Staubli VAL3: recvHeartbeat.pgx

public program recvHeartbeat()
  local num l_nByte
  local num l_nBytesRecv
  local num l_nHtbt
  local num l_nHtbtB[4]
  local num l_nIndex
begin
  while (true)
    l_nBytesRecv=0
    l_nIndex=0
    // if heartbeat is expected (used with mock client)
    if (bCheckHeartbeat)
      // attempt to receive heartbeat
      while (l_nBytesRecv<4)
        l_nIndex=sioGet(siTcpIpFbk,l_nByte)
        if (l_nIndex==1)
          l_nHtbtB[l_nBytesRecv]=l_nByte
          l_nBytesRecv=l_nBytesRecv+l_nIndex
        elseIf (l_nIndex==-1)
          // error or timeout, indicate only if connection previously established
          if (nDataOut==1)
            nDataOut=-1
            // close connection properly (to avoid CLOSE_WAIT)
            clearBuffer(siTcpIpFbk)
          endIf
        endIf
      endWhile
      // received 4 bytes
      l_nIndex=fromBinary(l_nHtbtB,4,"-4l",l_nHtbt)
      if (l_nIndex==1)
        // confirm heartbeat value -> ensure it is connected
        if (l_nHtbt==11002)
          nDataOut=1
        endIf
      endIf
    else
      // no heartbeat is expected (used with generic industrial_robot_client)
      l_nIndex = sioGet(siTcpIpFbk, l_nByte)
      if (l_nIndex == -1)
        // connection not established or connection lost
        if (nDataOut == 1)
          nDataOut = -1
        endIf
      else
        // it means l_nIndex >= 0: connection established
        if (nDataOut == 0)
          // delay data output to avoid sync issues with client
          delay(1.0)
        endIf
        // flag connection as established
        nDataOut = 1
      endIf
    endIf
  endWhile
end
